// TIA Portal V16 export
// export: Created 2021-07-12T14:47:20.955961Z, ExportSetting WithDefaults, DisplayName Totally Integrated Automation Portal, DisplayVersion V16, DisplayName TIA Portal Version Control Interface, DisplayVersion V16, DisplayName TIA Portal Openness, DisplayVersion V16, DisplayName STEP 7 Professional, DisplayVersion V16, DisplayName STEP 7 Safety, DisplayVersion V16, DisplayName WinCC Professional, DisplayVersion V16
TYPE "SimaHydTO_typeHMIConnectionVCharEditorParameter"
TITLE = SimaHydTO_typeHMIConnectionVCharEditorParameter
// HMI interface: VChar editor
// stored: IsFailsafeCompliant false
   STRUCT
      ActualTableStartIndex : Int;
      SelectedTableIndex : Int;
      MaximumNumberOfLines : Int;
      NumberOfUsedLines : Int;
      NumberOfUsableLines : Int;
   END_STRUCT;
END_TYPE
